FUNCTION_BLOCK TEST_ENDPOINT
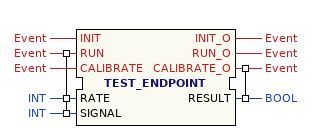
  EVENT_INPUT
    INIT;
    RUN WITH RATE, SIGNAL;
    CALIBRATE; {SET_ATTRIBUTE(OpcUa, Method)}
  END_EVENT
  EVENT_OUTPUT
    INIT_O;
    RUN_O;
    CALIBRATE_O WITH RESULT;
  END_EVENT
  VAR_INPUT
    RATE : INT; {SET_ATTRIBUTE(OpcUa, Constant)}
    SIGNAL : INT; {SET_ATTRIBUTE(OpcUa, Variable)}
  END_VAR
  VAR_OUTPUT
    RESULT : BOOL; {SET_ATTRIBUTE(OpcUa, CALIBRATE)}
  END_VAR
END_FUNCTION_BLOCK
(* other elements stored in the file *)
(* SelfDescription FBType=POINT.ENDPOINT *)
